TYPE EL4024_HWTOPLC_PDOS :
	STRUCT
		
	
	Channel1 	AT %Q* : INT;
	Channel2 	AT %Q* : INT;
	Channel3 	AT %Q* : INT;
	Channel4 	AT %Q* : INT;

	END_STRUCT
END_TYPE

(* stored: Version 1.1.0.1, ProductVersion 3.1.4024.15
   DUT EL4024_HWTOPLC_PDOS: Id {af59b89d-8491-4340-af99-4d2569832420} *)
